FUNCTION_BLOCK PUBLIC FB_Light IMPLEMENTS I_Light
VAR_INPUT
	bOn					:	BOOL;
	bOff				:	BOOL;
END_VAR
VAR_OUTPUT
	bControl			:	BOOL;
END_VAR
VAR
	rtrigOn				:	R_TRIG;
	rtrigOff			:	R_TRIG;
	_bControlLevel		:	BOOL;
END_VAR

rtrigOn(CLK := bOn);
IF (rtrigOn.Q) THEN
	M_On();
END_IF

rtrigOff(CLK := bOff);
IF (rtrigOff.Q) THEN
	M_Off();
END_IF

bControl := bControlLevel;

METHOD PUBLIC M_On
_bControlLevel := TRUE;
END_METHOD

PROPERTY bControlLevel : BOOL
SET
END_SET
GET
bControlLevel := _bControlLevel;
END_GET
END_PROPERTY

METHOD PUBLIC M_Off
_bControlLevel := FALSE;
END_METHOD

END_FUNCTION_BLOCK

(* stored: Version 1.1.0.1, ProductVersion 3.1.0.23
   POU FB_Light: Id {ac651da5-5748-4f92-a579-c38eff465f2e}
   Method M_On: Id {0b05d84c-3c99-44b7-a9f9-a9a6e37e56c6}
   Property bControlLevel: Id {8f0a6793-97a1-42fb-89c5-c7cbe36a5815}
   Set Set: Id {757bccf7-c33a-4e19-8fa3-ae6d57cc983b}
   Get Get: Id {8452bba2-c009-4ca5-b8e7-8e3bfd4cda70}
   Method M_Off: Id {cd28f873-04eb-42ed-b680-18b8c9700ed2} *)
